{attribute addProperty BoxType "EL2878-0005-0016"}
{attribute addProperty Id "DiagnosticAT %I*Diagnostic_4CD4E3A2810ChannelAT %Q*ARRAY[0..7] OF Channel_7F374EB06480WcStateAT %I*WcState_F855686C1620InfoDataAT %I*InfoData_192954DE1620"}
{attribute addProperty CRC "2999521889"}
{attribute addProperty SizeInBites "104"}
{attribute addProperty SizeInBytes "13"}
TYPE EL2878_4C8AEF8F :
STRUCT
	{attribute addProperty Name "Diagnostic"}
	Diagnostic : Diagnostic_4CD4E3A2;
	{attribute addProperty Name "Channel"}
	Channel : ARRAY[0..7] OF Channel_7F374EB0;
	{attribute addProperty Name "WcState"}
	WcState : WcState_F855686C;
	{attribute addProperty Name "InfoData"}
	InfoData : InfoData_192954DE;
END_STRUCT
END_TYPE

(* stored: Version 1.2.0.0, ProductVersion 3.1.4024.9
   DUT EL2878_4C8AEF8F: Id {c868b786-a916-4982-86ba-870bf82403ef} *)
